// TIA Portal V17 export
// export: Created 2025-03-07T09:19:08.8833624Z, ExportSetting WithDefaults, DisplayName Totally Integrated Automation Portal, DisplayVersion V17 Update 8, DisplayName TIA Portal Openness, DisplayVersion V17 Update 8, DisplayName TIA Portal Version Control Interface, DisplayVersion V17, DisplayName SINAMICS Startdrive Advanced, DisplayVersion V17 SP2, DisplayName SINAMICS Startdrive G110M, G120, G120C, G120D, G120P, G115D, DisplayVersion V17 SP2, DisplayName SINAMICS Startdrive G130, G150, S120, S150, SINAMICS MV, S210, DisplayVersion V17 SP2, DisplayName STEP 7 Professional, DisplayVersion V17 Update 8, DisplayName SINUMERIK ONE STEP 7 Toolbox, DisplayVersion V17 Update 12, DisplayName SINUMERIK 840D sl STEP 7 Toolbox, DisplayVersion V17 Update 12, DisplayName STEP 7 Safety, DisplayVersion V17 Update 6, DisplayName WinCC Advanced, DisplayVersion V17 Update 8
FUNCTION "FC7200_HMI_FUNCTION" : Void   // FC7200, LAD
{ S7_Optimized_Access := 'FALSE' }
AUTHOR : ETXETAR
VERSION : 1.0
// stored: AutoNumber false, IsIECCheckEnabled false, SetENOAutomatically false, UDAEnableTagReadback false
   VAR_TEMP
      SCREEN_NAV : Bool;   // SCREEN NAVEGATION OPTION
      CNC_STATUS : Bool;   // CNC STATUS OPTION
      X : Int;
   END_VAR
   VAR CONSTANT
      TOTAL_SCREEN_NUM : Int := 89;
      FC_NUMBER : DInt := 7200;
   END_VAR
BEGIN

REGION Network 1: OPTIONS OFF
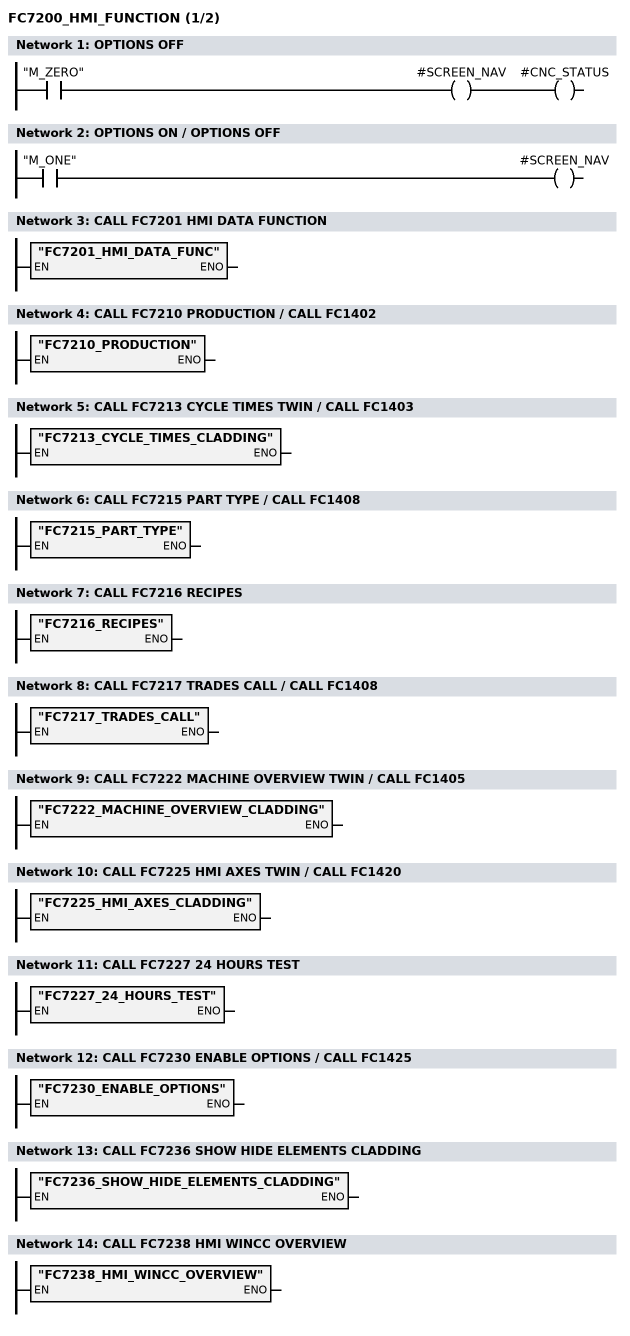
   RUNG wire#powerrail
      Contact( "M_ZERO" )
      Coil( #SCREEN_NAV )
      Coil( #CNC_STATUS )
   END_RUNG
   // the same network as SCL:
   #SCREEN_NAV := "M_ZERO";
   #CNC_STATUS := "M_ZERO";
END_REGION

REGION Network 2: OPTIONS ON / OPTIONS OFF
   RUNG wire#powerrail
      Contact( "M_ONE" )
      Coil( #SCREEN_NAV )
   END_RUNG
   // the same network as SCL:
   #SCREEN_NAV := "M_ONE";
END_REGION

REGION Network 3: CALL FC7201 HMI DATA FUNCTION
   RUNG wire#powerrail
      "FC7201_HMI_DATA_FUNC"()
   END_RUNG
   // the same network as SCL:
   "FC7201_HMI_DATA_FUNC"();
END_REGION

REGION Network 4: CALL FC7210 PRODUCTION / CALL FC1402
   RUNG wire#powerrail
      "FC7210_PRODUCTION"()
   END_RUNG
   // the same network as SCL:
   "FC7210_PRODUCTION"();
END_REGION

REGION Network 5: CALL FC7213 CYCLE TIMES TWIN / CALL FC1403
   RUNG wire#powerrail
      "FC7213_CYCLE_TIMES_CLADDING"()
   END_RUNG
   // the same network as SCL:
   "FC7213_CYCLE_TIMES_CLADDING"();
END_REGION

REGION Network 6: CALL FC7215 PART TYPE / CALL FC1408
   RUNG wire#powerrail
      "FC7215_PART_TYPE"()
   END_RUNG
   // the same network as SCL:
   "FC7215_PART_TYPE"();
END_REGION

REGION Network 7: CALL FC7216 RECIPES
   RUNG wire#powerrail
      "FC7216_RECIPES"()
   END_RUNG
   // the same network as SCL:
   "FC7216_RECIPES"();
END_REGION

REGION Network 8: CALL FC7217 TRADES CALL / CALL FC1408
   RUNG wire#powerrail
      "FC7217_TRADES_CALL"()
   END_RUNG
   // the same network as SCL:
   "FC7217_TRADES_CALL"();
END_REGION

REGION Network 9: CALL FC7222 MACHINE OVERVIEW TWIN / CALL FC1405
   RUNG wire#powerrail
      "FC7222_MACHINE_OVERVIEW_CLADDING"()
   END_RUNG
   // the same network as SCL:
   "FC7222_MACHINE_OVERVIEW_CLADDING"();
END_REGION

REGION Network 10: CALL FC7225 HMI AXES TWIN / CALL FC1420
   RUNG wire#powerrail
      "FC7225_HMI_AXES_CLADDING"()
   END_RUNG
   // the same network as SCL:
   "FC7225_HMI_AXES_CLADDING"();
END_REGION

REGION Network 11: CALL FC7227 24 HOURS TEST
   RUNG wire#powerrail
      "FC7227_24_HOURS_TEST"()
   END_RUNG
   // the same network as SCL:
   "FC7227_24_HOURS_TEST"();
END_REGION

REGION Network 12: CALL FC7230 ENABLE OPTIONS / CALL FC1425
   RUNG wire#powerrail
      "FC7230_ENABLE_OPTIONS"()
   END_RUNG
   // the same network as SCL:
   "FC7230_ENABLE_OPTIONS"();
END_REGION

REGION Network 13: CALL FC7236 SHOW HIDE ELEMENTS CLADDING
   RUNG wire#powerrail
      "FC7236_SHOW_HIDE_ELEMENTS_CLADDING"()
   END_RUNG
   // the same network as SCL:
   "FC7236_SHOW_HIDE_ELEMENTS_CLADDING"();
END_REGION

REGION Network 14: CALL FC7238 HMI WINCC OVERVIEW
   RUNG wire#powerrail
      "FC7238_HMI_WINCC_OVERVIEW"()
   END_RUNG
   // the same network as SCL:
   "FC7238_HMI_WINCC_OVERVIEW"();
END_REGION

REGION Network 15 (SCL): SCREEN NAVIGATION

       IF #SCREEN_NAV THEN
           FOR #X := 11 TO #TOTAL_SCREEN_NUM DO
               IF "DB7200_HMI_FUNCTION".SCREEN_SELECTION[#X] THEN
                   "DB7200_HMI_FUNCTION".PLC_SCREEN_SELECTION :=INT_TO_WORD(#X);
               END_IF;
           END_FOR;
       END_IF;
END_REGION

REGION Network 16: CNC STATUS
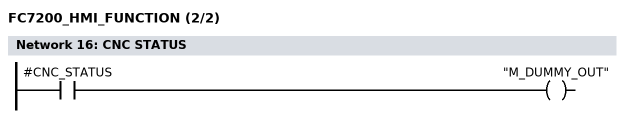
   RUNG wire#powerrail
      Contact( #CNC_STATUS )
      Coil( "M_DUMMY_OUT" )
   END_RUNG
   // the same network as SCL:
   "M_DUMMY_OUT" := #CNC_STATUS;
END_REGION
END_FUNCTION
